{attribute 'qualified_only'}
VAR_GLOBAL CONSTANT
	RED_GREEN_LIGHT_INTERVAL : TIME := T#5000MS;
	YELLOW_LIGHT_INTERVAL : TIME := T#1000MS;
	FLASHING_YELLOW_LIGHT_INTERVAL : TIME := T#1000MS;

	MIN_LIGHT_SWITCH_SPEED_CORECTION_PERCENT : SINT := -30;	
	MAX_LIGHT_SWITCH_SPEED_CORECTION_PERCENT : SINT := +30;	

	TRAFFIC_LIGHTS_PER_GROUP : BYTE := 2;
	TOTAL_TRAFFIC_LIGHTS : BYTE := TRAFFIC_LIGHTS_PER_GROUP * 2;
END_VAR

(* stored: Version 1.1.0.1
   GVL IntersectionConstants: Id {83aeeddc-5029-4f41-bce3-e0ecb481deb2} *)
